// TIA Portal V16 export
// export: Created 2023-02-02T16:29:09.1406952Z, ExportSetting WithDefaults, DisplayName Totally Integrated Automation Portal, DisplayVersion V16 Update 3, DisplayName TIA Portal Version Control Interface, DisplayVersion V16 Update 2, DisplayName TIA Portal Openness, DisplayVersion V16 Update 3, DisplayName STEP 7 Professional, DisplayVersion V16 Update 3, DisplayName STEP 7 Safety, DisplayVersion V16, DisplayName WinCC Professional, DisplayVersion V16 Update 3
DATA_BLOCK "DB31101_Dy_DevValveBi"   // DB31101
TITLE = Dynamic DB [DEVICE DRIVER] — Bistable Valve
{ S7_Optimized_Access := 'TRUE' }
AUTHOR : M_Gledhill
FAMILY : DeviceDriver
NAME : Dy_DevValveBi
VERSION : 1.0
// PRACTICAL SERIES AUTOMATION LIBRARY (PAL)   —   COPYRIGHT 2020 – M. GLEDHILL (MIT LICENCE)
//                   ———— ◆ ————
// FULL ONLINE DOCUMENTATION IS AVAILABLE AT: https://practicalseries.com/2001-pal/index.html
// stored: AutoNumber false, DBAccessibleFromOPCUA true, IsOnlyStoredInLoadMemory false, IsRetainMemResEnabled false, IsWriteProtectedInAS false, MemoryReserve 100
   VAR
      _DB_Header { ExternalAccessible := 'False'; ExternalVisible := 'False'; ExternalWritable := 'False'} : Array[0..79] of Bool;   // Dynamic DB [DEVICE DRIVER] — Bistable Valve
      __________0000_0 { ExternalAccessible := 'False'; ExternalVisible := 'False'; ExternalWritable := 'False'} : Bool := false;
      __________0000_1 { ExternalAccessible := 'False'; ExternalVisible := 'False'; ExternalWritable := 'False'} : Bool := false;   // ▀▀▀▀ DB CURRENT REVISION
      revInfo { ExternalWritable := 'False'; S7_SetPoint := 'True'} : "UT01000_St_SysRevision";   // Revision information
      __________0010_0 { ExternalAccessible := 'False'; ExternalVisible := 'False'; ExternalWritable := 'False'} : Bool := false;
      __________0010_1 { ExternalAccessible := 'False'; ExternalVisible := 'False'; ExternalWritable := 'False'} : Bool := false;   // ▀▀▀▀ ISOLATING VALVES
      V001 { ExternalWritable := 'False'} : "UT31101_Dy_DevValveBi";   // Filter 1 backwash inlet
   END_VAR
BEGIN
   // _DB_Header[0] : ▄▄▄▄▄▄▄▄▄▄▄▄▄▄▄▄▄▄▄▄▄▄▄▄▄▄▄▄▄▄▄▄▄ ＳＴＡＮＤＡＲＤ ▄▄
   // _DB_Header[2] : TITLE: DEVICE DRIVER — BISTABLE VALVE
   // _DB_Header[4] : ▀▀▀▀▀▀▀▀▀▀▀▀▀▀▀▀▀▀▀▀▀▀▀▀▀▀▀▀▀▀▀▀▀▀▀▀▀▀▀▀▀▀▀▀
   // _DB_Header[5] : TYPE: DYNAMIC
   // _DB_Header[6] : ▄▄▄▄▄▄▄▄▄▄▄▄▄▄▄▄▄▄▄▄▄▄▄▄▄▄▄▄▄▄▄▄▄▄▄▄▄▄▄▄▄▄▄▄
   // _DB_Header[8] : This is the dynamic data block associated with the standard device driver for an isolating valve
   // _DB_Header[9] : block:
   // _DB_Header[10] : FC11101_StdDevValveBi
   // _DB_Header[12] : The dynamic data holds the live data for the device (its mode, status and messages
   // _DB_Header[13] : and any other dynamic information required by the module)
   // _DB_Header[15] : Each valve is given the user data type:
   // _DB_Header[16] : UT31101_Dy_DevValveBi
   // _DB_Header[17] : This holds the full set of dynamic data for the device
   // _DB_Header[19] : ━━━ ⬙⬙⬙⬙⬙⬙ ━━━
   // _DB_Header[21] : ▄▄▄▄▄▄▄▄▄▄▄▄▄▄▄▄▄▄▄▄▄▄▄▄▄▄▄▄▄▄▄▄▄▄▄▄▄▄▄▄▄▄▄▄
   // _DB_Header[22] : MODIFICATION HISTORY
   // _DB_Header[24] : This is a summary of the recent software modifications made to this block (most recent at top)
   // _DB_Header[26] : ―――――――――――――――――――――――――――――――――――――――――――
   // _DB_Header[27] : DATE REVISION MASTER BRANCH DEV
   // _DB_Header[28] : (nnn.amm) COMMIT TAG (Base ---> Merge) BRANCH Author
   // _DB_Header[29] : ———————————————————————————————————————————
   // _DB_Header[30] : 2023.02.02 001.000 D0016 D0015 D0016 None M. Gledhill
   // _DB_Header[31] : FC11101 — RELEASED FOR USE
   // _DB_Header[32] : Merge back to master branch
   // _DB_Header[34] : 2023.02.01 000.801 D0015A-000.801 D0015 N/A D0015A M. Gledhill
   // _DB_Header[35] : FC11101 — Released for test (SMTS)
   // _DB_Header[37] : 2023.01.28 000.102 D0015A-000.102 D0015 N/A D0015A M. Gledhill
   // _DB_Header[38] : FC11101 — Incremental build
   // _DB_Header[40] : 2022.08.15 000.101 D0015A-000.101 D0008 N/A D0015A M. Gledhill
   // _DB_Header[41] : FC11101 Block created
   // _DB_Header[42] : ———————————————————————————————————————————
   // _DB_Header[43] : Where: nnn = Major revision
   // _DB_Header[44] : a = Type (1-7 Development, 8 Proving, 9 Qualification, 0 Release)
   // _DB_Header[45] : mm = Minor revision (must be 00 if a = 0)
   // _DB_Header[46] : Block properties version number should be set to nn.a (only one decimal place)
   // _DB_Header[48] : ██████████████ █ █ █ █ END █ █ █ █ ██████████████
   revInfo.REV_BLOCK := 'DB31101';
   revInfo.REV_NUMBER := '001.000';
   revInfo.REV_DATE := '2023.02.02';
   revInfo.REV_AUTHOR := 'M. Gledhill';
END_DATA_BLOCK
